FUNCTION_BLOCK fb_prod_rate_ctrl

VAR_INPUT
	kc: REAL;
	ti:REAL;
	ts:REAL;
	hi:REAL;
	lo:REAL;
	x0:REAL := 0;
	set_prod_rate: REAL := g_set_production;
	//xmv17: REAL;

END_VAR

VAR_OUTPUT
	Prodsp: REAL := 0;
	Fp: REAL :=0;
END_VAR

VAR
	
	vel_p: fb_vel_pi;
	x: FB_CTRL_2POINT;
	zoh_real_0: fb_zoh_real := (xlast := x0 );
	change_rate_limit: FB_CTRL_LIMITER := (stInternalParams := (fMinOutput := -0.286875, fMaxOutput := 0.286875));
	rate: REAL := 0;
	
	prodsp_scaled: REAL;
	calc_change_rate: FB_CTRL_D;
	integrate_change_rate: FB_CTRL_I;
	prod_rate_saturate: FB_CTRL_LIMITER;
	prod_rate_saturate_params: ST_CTRL_LIMITER_PARAMS := (fMinOutput := lo, fMaxOutput := hi);
	last_prod_rate: REAL := 0.0;
	
	stparams_calc_change_rate: ST_CTRL_D_PARAMS;
	stparams_change_rate_limit: ST_CTRL_LIMITER_PARAMS;
	stparams_integrate_change_rate: ST_CTRL_I_PARAMS;
	
END_VAR

VAR CONSTANT
	ProdspGain: REAL := 100/22.89;
END_VAR

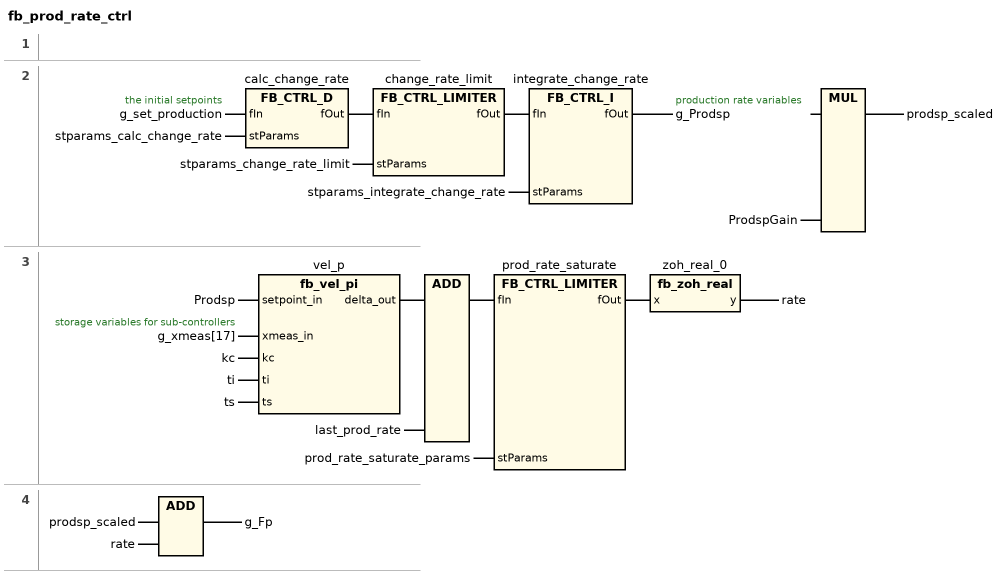
// NETWORK 1

// NETWORK 2
//   g_set_production: the initial setpoints
//   g_Prodsp: production rate variables
calc_change_rate(fIn := g_set_production, stParams := stparams_calc_change_rate); // FB_CTRL_D
change_rate_limit(fIn := calc_change_rate.fOut, stParams := stparams_change_rate_limit); // FB_CTRL_LIMITER
integrate_change_rate(fIn := change_rate_limit.fOut, stParams := stparams_integrate_change_rate); // FB_CTRL_I
g_Prodsp := integrate_change_rate.fOut;
prodsp_scaled := integrate_change_rate.fOut * ProdspGain;

// NETWORK 3
//   g_xmeas[17]: storage variables for sub-controllers
vel_p(setpoint_in := Prodsp, xmeas_in := g_xmeas[17], kc := kc, ti := ti, ts := ts); // fb_vel_pi
prod_rate_saturate(fIn := vel_p.delta_out + last_prod_rate, stParams := prod_rate_saturate_params); // FB_CTRL_LIMITER
zoh_real_0(x := prod_rate_saturate.fOut); // fb_zoh_real
rate := zoh_real_0.y;

// NETWORK 4
g_Fp := prodsp_scaled + rate;

END_FUNCTION_BLOCK

(* stored: Version 1.1.0.1, ProductVersion 3.1.0.26
   POU fb_prod_rate_ctrl: Id {12afc640-1cc9-456e-b128-0a54a95b7ca0} *)
